INTERFACE ITcMessage_Ext

METHOD Send : BOOL
VAR_INPUT
	eventType : Tc3_EventLogger.TcEventEntry;
	args : STRING(255);
END_VAR
END_METHOD

END_INTERFACE

(* stored: Version 1.1.0.1, ProductVersion 3.1.4024.11
   Itf ITcMessage_Ext: Id {ecc02940-e99f-4b59-aa27-20f74ac0a53f}
   Method Send: Id {974ef709-63a5-449e-b808-feae03cbbc39} *)
